(* CoDeSys 2.3 export: GetStringLength.EXP *)

(* POU MQTT-Utils/GetStringLength, ST *)
FUNCTION GetStringLength : UINT
VAR_INPUT
	pString			: POINTER TO BYTE;
END_VAR
VAR
END_VAR
GetStringLength := 0;
WHILE pString^ <> 0 DO
	pString := pString + 1;
	GetStringLength := GetStringLength + 1;
END_WHILE
END_FUNCTION
